// TIA Portal V20 export
TYPE "zp_CITI_Parameters"
// stored: Access Published, Namespace CITI_Logic
   STRUCT
      Map_ID : SInt;
      MachineType : SInt;
      Rtd_CycTime : DInt := 0;
      Flt_Det_Dly : Int := 0;
      DTT_IN : Int;
      DTT_OUT : Int;
      CycTime_DataDly : DInt := 0;
      CycleTime_Data_Dwll : DInt := 0;
      Parts_Per_Cyc : Int := 0;
      RetryCnt : Int := 0;
      FlasherRate : Int := 0;
   END_STRUCT;
END_TYPE
